// TwinCAT 3 PLC project PLC1
// ProgramVersion: 3.1.4026.25
// libraries:
//   Tc2_Standard, * (Beckhoff Automation GmbH)
//   Tc2_System, * (Beckhoff Automation GmbH)
//   Tc3_Module, * (Beckhoff Automation GmbH)
// project tree:
//   Diagrams/ Class Diagram.TcCD (not stored)
//   FBs/ FB_LAMP_DIMM.TcPOU (not stored), FB_LAMP_ONOFF.TcPOU
//   ITFs/ I_LampCtrl.TcIO (not stored)
//   / PlcTask.TcTTO
//   POUs/ MAIN.TcPOU
// real-time tasks:
//   TASK PlcTask: cycle T#10ms, priority 20, ADS port 350

CONFIGURATION PLC1
    RESOURCE PLC ON TwinCAT3
        TASK PlcTask(INTERVAL := T#10ms, PRIORITY := 20);
        PROGRAM MAIN WITH PlcTask : MAIN;
    END_RESOURCE
END_CONFIGURATION

// ---- POUs/MAIN.TcPOU
PROGRAM MAIN
VAR
	// Used to demo ITF reference on start-up
	fbLamp1 	: FB_LAMP_DIMM;
	fbLamp2 	: FB_LAMP_ONOFF;
	
	
	// Interface
	LampCtrl 	: ARRAY[0..1] OF I_LampCtrl := [fbLamp1, fbLamp2];
	
	// Program Control
	bLightsOn	: BOOL;
	bLightsOff	: BOOL;
	State		: ARRAY[0..1] OF STRING;
END_VAR

IF bLightsOn THEN
	IF LampCtrl[0].ON() AND LampCtrl[1].ON() THEN
		bLightsOn := FALSE;
	END_IF
END_IF

IF bLightsOff THEN	
	IF LampCtrl[0].OFF() AND LampCtrl[1].OFF() THEN
		bLightsOff := FALSE;
	END_IF
END_IF

State[0] := LampCtrl[0].State;
State[1] := LampCtrl[1].State;

END_PROGRAM

// ---- FBs/FB_LAMP_ONOFF.TcPOU
{attribute 'reflection'}
FUNCTION_BLOCK FB_LAMP_ONOFF IMPLEMENTS I_LampCtrl
VAR_INPUT
END_VAR
VAR_OUTPUT
END_VAR
VAR
	bOutHw AT%Q*:BOOL;
	
	{attribute 'instance-path'}
	{attribute 'no_init'}
	sPath: STRING;
END_VAR

METHOD OFF : BOOL
// implementation switch Lamp off
OFF := FALSE;

bOutHw := FALSE;
OFF := TRUE;
END_METHOD

METHOD ON : BOOL
// implementation switch Lamp on
ON := FALSE;

bOutHw := TRUE;
ON := TRUE;
END_METHOD

PROPERTY State : string
GET
// additional demo pathname of FB
State := CONCAT('Object: ', sPath); 
State := CONCAT(State, 'State:'); 
State := CONCAT(State, BOOL_TO_STRING(bOutHw));
END_GET
END_PROPERTY

END_FUNCTION_BLOCK
